{attribute 'qualified_only'}
VAR_GLOBAL
	// Rezept-Controlword
	{attribute 'OPC.UA.DA' := '1'}
	CW		:RezeptControlWord;
	
	// Rezept-Statusword
	{attribute 'OPC.UA.DA' := '1'}
	SW		:RezeptStatusWord;
END_VAR

(* stored: Version 1.1.0.1, ProductVersion 3.1.4024.12
   GVL GVL_OPC_UA: Id {30465ce4-cb68-4b5b-899c-6742322bd070} *)
